RoboDK station: Pick_And_Place_Chapter.rdk

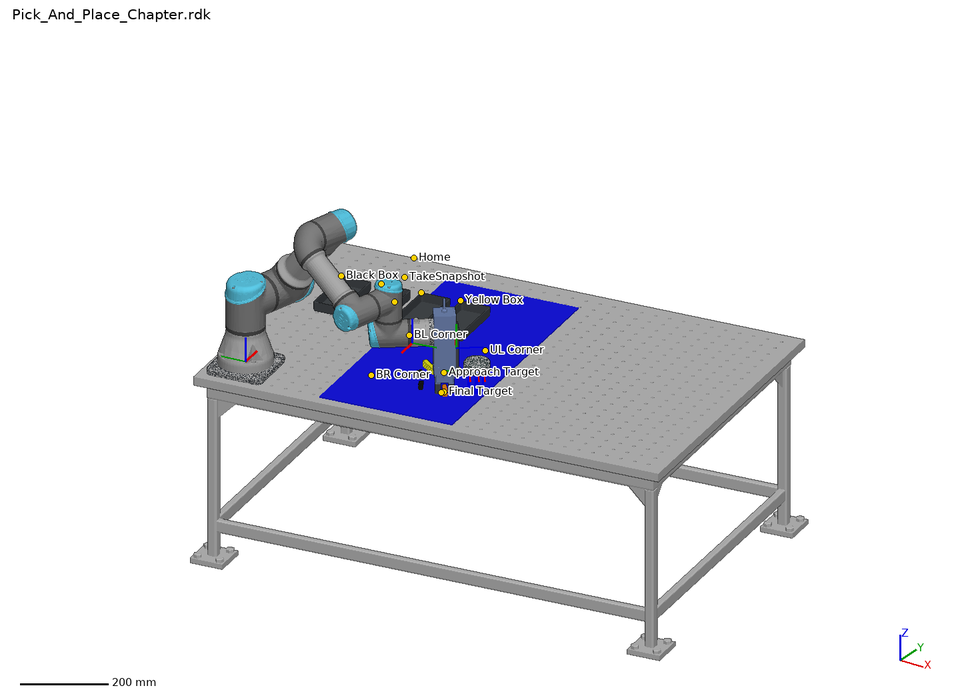
[picture v0: the station drawn from its stored meshes, robots at their saved joint values, targets as dots, program paths as lines]
Station Pick_And_Place_Chapter (saved by RoboDK 5.6.0). Poses are relative to the parent item; angles as X-Y-Z fixed-axis rotations.
Station parameters (name, value as stored): IO_1, 0, IO_0, 0, IO_10, CollisionFreePlanner, UR3e, CollisionFreePlanner-Rob UR3e
  - frame UR3e Base at (0, 0, 0) mm, rotated rx 0 ry 0 rz 99.55 deg
    - robot UR3e: 6 axes, payload 3 kg, reach 500 mm, repeatability 0.03 mm, weight 11 kg
        modified DH rows (alpha deg, a mm, theta deg, d mm): 0, 0, 0, 151.9; 90, 0, 180, 0; 0, 243.55, 0, 0; 0, 213.2, 0, 131.05; -90, 0, 0, 85.35; 90, 0, 180, 92.1
        joint limits [-45, -150, 0, -150, -150, -200] to [180, 90, 160, 90, 165, -160]; home [0, -90, -90, 0, 90, 0]; saved at [69.529, -51.763, 84.677, -32.914, 39.801, -180]
      - frame Cam L515 at (0, 100, 90.15) mm, rotated rx -90 ry 0 rz 0 deg
        - frame L515 RGB Cam at (0, 0, 0) mm
          - camera Camera_rgb
        - frame L515 Depth Cam at (0, 0, 0) mm, rotated rx 0.31 ry 0 rz 0 deg
          - camera Camera_depth
        - object Intel_RealSense_L515_Housing_reduced at (0, -18.82, 0) mm, rotated rx 0 ry 0 rz 180 deg, size 61 x 60.7 x 26 mm, geometry from Intel_RealSense_L515_Housing_reduced.stp
      - frame Cam L515 real at (0, 100, 106.15) mm, rotated rx -90 ry 0 rz 0 deg
      - tool RGI14_cBrida_UR3e_turnedFingers, TCP at (0, 153, 35) mm, rotated rx 0 ry 90 rz 90 deg, size 63 x 236.5 x 60 mm, geometry from RGI14_cBrida_UR3e_turnedFingers.stp
      - tool RGI14_cBrida_UR3e, TCP at (0, 153, 35) mm, rotated rx -90 ry 0 rz 0 deg, size 63 x 236.5 x 60 mm, geometry from RGI14_cBrida_UR3e.stp
      - frame L515 real measured at (0, 100, 108.97) mm, rotated rx -90 ry 0 rz 0 deg
      - frame L515 rgb sensor at (0.04, 100, 122.97) mm, rotated rx -90 ry 0 rz 0 deg
      - frame Flange_camera at (0, 42.5, 63) mm, rotated rx 0 ry 0 rz 180 deg
        - object Brida_RGI14_L515 at (0, 0, 0) mm, size 50 x 115 x 6 mm, geometry from Brida_RGI14_L515.stp
    - target Home (Cartesian target) at (233, -312.03, 223.29) mm, rotated rx 180 ry 0 rz 90 deg; joints [115.423, -73.84, 53.012, 20.829, 115.423, -180] of UR3e
    - object Table at (-50, -125, -15) mm, size 333.2 x 666.5 x 3.3 mm, geometry from Table.stp
    - target TakeSnapshot (Cartesian target) at (255.94, -277.09, 157.08) mm, rotated rx -179.99 ry 0 rz 135 deg; joints [100.001, -89.997, 89.999, 0.002, 54.999, -180.014] of UR3e
    - target Final Target (Cartesian target) at (70.49, -465.1, -11) mm, rotated rx -180 ry 0 rz -150.27 deg; joints [134.995, -90.002, 90.379, 179.62, -89.999, 359.992] of UR3e
    - target Approach Target (Cartesian target) at (70.49, -465.1, 39) mm, rotated rx -180 ry 0 rz -150.27 deg; joints [101.326, 342.717, 17.958, -0.674, -13.669, -180] of UR3e
    - target Yellow Box (Cartesian target) at (400, -350, 50) mm, rotated rx 180 ry -0.01 rz 180 deg; joints [110.773, -29.744, 25.537, 4.235, 20.773, -180.026] of UR3e
    - object Yellow Box at (400, -350, -15) mm, size 150 x 75 x 25 mm, geometry from Box.stp
    - target Black Box (Cartesian target) at (400, -50, 50) mm, rotated rx 180 ry -0.01 rz 180 deg; joints [141.435, -76.58, 104.682, -28.09, 51.435, -180.008] of UR3e
    - object Black Box at (400, -50, -15) mm, size 150 x 75 x 25 mm, geometry from Box.stp
    - target Orange Box (Cartesian target) at (400, -150, 50) mm, rotated rx 180 ry -0.01 rz 180 deg; joints [126.322, -68.486, 93.487, -24.985, 36.322, -180.014] of UR3e
    - object Orange Box at (400, -150, -15) mm, size 150 x 75 x 25 mm, geometry from Box.stp
    - target White Box (Cartesian target) at (400, -250, 50) mm, rotated rx 180 ry -0.01 rz 180 deg; joints [116.774, -54.333, 71.069, -16.714, 26.774, -180.02] of UR3e
    - object White Box at (400, -250, -15) mm, size 150 x 75 x 25 mm, geometry from Box.stp
    - target BR Corner (Cartesian target) at (31.84, -301.17, 14.98) mm, rotated rx -179.99 ry 0.01 rz 90.74 deg; joints [51.971, -100.389, 140.773, -40.391, 51.232, -180.007] of UR3e
    - target UR Corner (Cartesian target) at (17.56, -482.51, 15) mm, rotated rx -179.99 ry 0.01 rz 90.74 deg; joints [70.955, -54.633, 81.745, -27.118, 70.216, -180.009] of UR3e
    - target UL Corner (Cartesian target) at (255.49, -479.44, 14.96) mm, rotated rx -179.99 ry 0.01 rz 90.74 deg; joints [108.211, -33.393, 42.202, -8.814, 107.472, -180.012] of UR3e
    - target BL Corner (Cartesian target) at (253.04, -289.73, 14.94) mm, rotated rx -179.99 ry 0.01 rz 90.74 deg; joints [121.152, -67.041, 102.234, -35.199, 120.413, -180.014] of UR3e
    - target Take Snap new (Cartesian target) at (131.05, -312.03, 157.1) mm, rotated rx 180 ry 0 rz 90 deg; joints [90, -96.664, 96.222, 0.442, 90, -180] of UR3e
  - object Table-1167x700x467mm at (73.52, 316.58, -20) mm, rotated rx 0 ry 0 rz 9.55 deg, size 1178.3 x 781.7 x 466.7 mm, geometry from Table-2000x1200x800mm.stl
  - object Mounting_Plate_UR3e at (-0.08, 0.32, -15) mm, rotated rx 1.24 ry 0.1 rz 9.55 deg, size 140 x 140 x 15 mm, geometry from Mounting_Plate_UR3e.stp
  - program TurnPos 2 (2 instructions, listed below)
  - program TurnPos 1 (2 instructions, listed below)
  - program Gripper closed (2 instructions, listed below)
  - program Gripper open (2 instructions, listed below)
  - frame BL Corner at (254.32, 296.67, 0) mm, rotated rx 0 ry 0 rz -80.45 deg
    - object lego3 at (173, 156, -10) mm, rotated rx 0 ry 0 rz 30 deg, size 32 x 11.2 x 16 mm, geometry from lego3.stp
    - object lego2 at (89, 145, -10) mm, rotated rx 0 ry 0 rz 155 deg, size 24 x 11.2 x 16 mm, geometry from lego2.stp
    - object lego4 at (77, 64, -10) mm, rotated rx 0 ry 0 rz 52 deg, size 48 x 11.2 x 16 mm, geometry from lego4.stp
    - object lego1 at (181, 112, -10) mm, rotated rx 0 ry 0 rz -162 deg, size 16 x 11.2 x 16 mm, geometry from lego1.stp
    - object lego1 at (123, 75, -10) mm, rotated rx 0 ry 0 rz -36 deg, size 16 x 11.2 x 16 mm, geometry from lego1.stp
  - program Move to Target (2 instructions, listed below)
  - program Move to Snapshot (2 instructions, listed below)
  - program Approach Target (1 instructions, listed below)
  - program Move to Home (1 instructions, listed below)
  - program Move to Black (2 instructions, listed below)
  - program Move to Yellow (2 instructions, listed below)
  - program Move to White (2 instructions, listed below)
  - program Move to Orange (2 instructions, listed below)
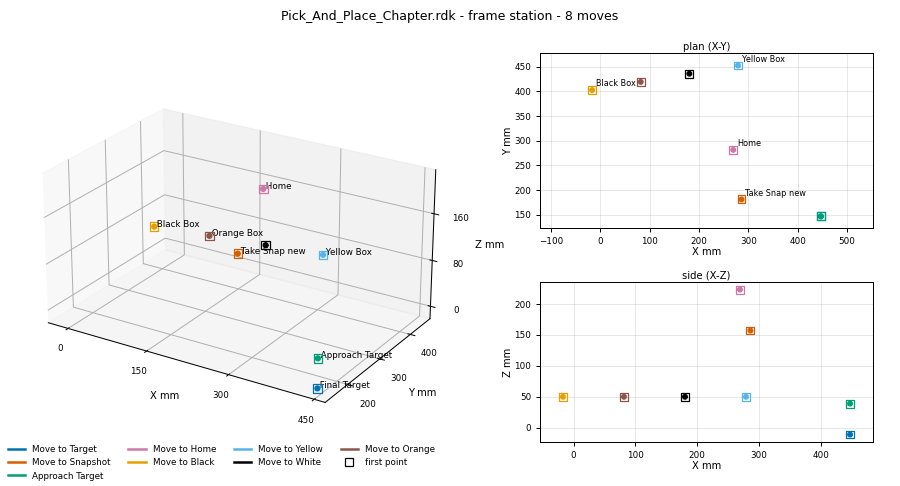
[picture p0: tool path of Pick_And_Place_Chapter.rdk in frame station, 8 of 8 moves have a stored position in this frame; points joined in program order, loops and branches not executed]

--- program TurnPos 2 (robot UR3e) ---
  Set IO_11=1
  Pause 1.0 s

--- program TurnPos 1 (robot UR3e) ---
  Set IO_11=0
  Pause 1.0 s

--- program Gripper closed (robot UR3e) ---
  Set IO_10=0
  Pause 1.0 s

--- program Gripper open (robot UR3e) ---
  Set IO_10=1
  Pause 1.0 s

--- program Move to Target (robot UR3e) ---
  MoveJ (Final Target)
  Pause 500 ms

--- program Move to Snapshot (robot UR3e) ---
  Set Tool: RGI14_cBrida_UR3e_turnedFingers
  MoveJ (Take Snap new)

--- program Approach Target (robot UR3e) ---
  MoveJ (Approach Target)

--- program Move to Home (robot UR3e) ---
  MoveJ (Home)

--- program Move to Black (robot UR3e) ---
  Set Tool: RGI14_cBrida_UR3e_turnedFingers
  MoveJ (Black Box)

--- program Move to Yellow (robot UR3e) ---
  Set Tool: RGI14_cBrida_UR3e_turnedFingers
  MoveJ (Yellow Box)

--- program Move to White (robot UR3e) ---
  Set Tool: RGI14_cBrida_UR3e_turnedFingers
  MoveJ (White Box)

--- program Move to Orange (robot UR3e) ---
  Set Tool: RGI14_cBrida_UR3e_turnedFingers
  MoveJ (Orange Box)
